FUNCTION IsBetween : BOOL
VAR_INPUT
	value: 	LREAL;
	minV:	LREAL;
	maxV:	LREAL;
END_VAR
VAR
END_VAR

IsBetween := value > minV AND value < maxV;

END_FUNCTION

(* stored: Version 1.1.0.1
   POU IsBetween: Id {068006e5-ff28-4dfb-8943-8706abd61fdb}, SpecialFunc None *)
